FUNCTION isLeapYear : Bool
VAR_INPUT
	nYear	: INT;
END_VAR
VAR
END_VAR

isLeapYear := (nYear / 4 = 0) AND (nYear / 100 <> 0) OR (nYear /400 = 0);

END_FUNCTION

(* stored: Version 1.1.0.1, ProductVersion 3.1.4024.11
   POU isLeapYear: Id {2336ce5d-2854-4e52-acb8-01e004829e85}, SpecialFunc None *)
